{attribute 'GeneratedUsingTerminal: EK1122-0000-0018'}
{attribute addProperty BoxType "EK1122-0000-0018"}
{attribute addProperty Id "Beckhoff_ELM36xxsub_EK1100EK1100_AB5A94672"}
{attribute addProperty CRC "2139685764"}
{attribute addProperty Size "2"}
TYPE Beckhoff_ELM36xxEK1122_7F890384 EXTENDS EK1122_AB5A9467 :
STRUCT
	{attribute addProperty Name "Beckhoff_ELM36xxsub_EK1100"}
	Beckhoff_ELM36xxsub_EK1100 : EK1100_AB5A9467;
END_STRUCT
END_TYPE

(* stored: Version 1.2.0.0, ProductVersion 3.1.4024.9
   DUT Beckhoff_ELM36xxEK1122_7F890384: Id {da7538d6-e2c7-43a2-8b65-889ebc18c807} *)
